{attribute 'OPC.UA.DA.StructuredType' := '1'}
FUNCTION_BLOCK FB_Sensor_IFM_PG2453 EXTENDS FB_BaseDevice IMPLEMENTS I_Device, I_Sensor

VAR

	{attribute 'OPC.UA.DA' := '0'} 
	eSensorType: E_SensorType;
	{attribute 'OPC.UA.DA' := '0'} 
	nRawInput AT %I*: INT;
	{attribute 'OPC.UA.DA' := '1'} 
	nCurrentValue: REAL;
	
	{attribute 'OPC.UA.DA' := '1'} 
	nVal4mA: REAL;
	{attribute 'OPC.UA.DA' := '1'} 
	nVal20mA: REAL;
END_VAR

calculate();

METHOD calculate : BOOL
VAR_INPUT
END_VAR
nCurrentValue := nVal4mA + (INT_TO_REAL(nRawInput) / GVL.nMaxADCOutput) * (nVal20mA - nVal4mA) ;
END_METHOD

{warning 'add method implementation '}
METHOD disable : BOOL
bEnable := FALSE;
END_METHOD

{warning 'add method implementation '}
METHOD enable : BOOL
bEnable := TRUE;
END_METHOD

{warning 'add method implementation '}
METHOD FB_init : BOOL
VAR_INPUT
	(* if TRUE, the retain variables are initialized (warm start / cold start)*)
	bInitRetains	: BOOL;
	(* if TRUE, the instance afterwards gets moved into the copy code (online change)*)
	bInCopyCode	: BOOL;
	SensorID	: STRING(80);
	SensorDescr	: STRING(255);
	SensorType	: E_SensorType;
	
END_VAR
sID := SensorID;
sDescr := SensorDescr;
eSensorType := SensorType;
END_METHOD

{warning 'add method implementation '}
METHOD getType : E_SensorType
getType := eSensorType;
END_METHOD

{warning 'add method implementation '}
METHOD getValue : REAL
getValue := nCurrentValue;
END_METHOD

METHOD setLimits : BOOL
VAR_INPUT
	Val_4mA: 	REAL;
	Val_20mA: 	REAL;
END_VAR
nVal4mA := Val_4mA;
nVal20mA := Val_20mA;
END_METHOD

{warning 'add method implementation '}
METHOD write : BOOL
END_METHOD

END_FUNCTION_BLOCK

(* stored: Version 1.1.0.1, ProductVersion 3.1.4024.12
   POU FB_Sensor_IFM_PG2453: Id {e52344af-298a-4608-abc5-bfd3e667bfc5}, SpecialFunc None
   Method calculate: Id {1a6eefaf-4812-4ec5-bf9b-fed404b7e71c}
   Method disable: Id {d8b03b0d-b8db-474a-8460-c337233d5e0f}
   Method enable: Id {e72ff0a2-45c3-4b55-897a-84897701f991}
   Method FB_init: Id {481cac8f-84a4-4fc8-9546-009268223c43}
   Method getType: Id {8a49c3d2-ec4b-4a0c-a523-a61eba544d43}
   Method getValue: Id {4eea110f-52d0-4f6a-9da9-7e256962e05f}
   Method setLimits: Id {6f417bbb-d5f4-47bf-8aec-ac943e0c5fe4}
   Method write: Id {17fe6040-b344-446b-b724-17730fb2f63b} *)
